FUNCTION_BLOCK PIDMgr3 (* Basic Function Block Type *)
  (* Standard: 61499-2 *)
  (* Version 0.0, 9/5/2025, Schneider Electric, Template *)
  PACKAGE SE.Nereda;
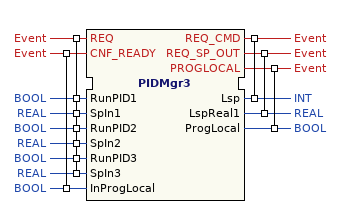
  EVENT_INPUT
    REQ WITH RunPID1, SpIn1, RunPID2, SpIn2, RunPID3, SpIn3; (* Normal Execution Request *)
    CNF_READY WITH InProgLocal;
  END_EVENT
  EVENT_OUTPUT
    REQ_CMD WITH Lsp;
    REQ_SP_OUT WITH LspReal1;
    PROGLOCAL WITH ProgLocal; (* Execution Confirmation *)
  END_EVENT
  VAR_INPUT
    RunPID1 : BOOL; (* Input event qualifier *)
    SpIn1 : REAL;
    RunPID2 : BOOL;
    SpIn2 : REAL;
    RunPID3 : BOOL;
    SpIn3 : REAL;
    InProgLocal : BOOL;
  END_VAR
  VAR_OUTPUT
    Lsp : INT;
    LspReal1 : REAL;
    ProgLocal : BOOL;
  END_VAR
  VAR
    InLsp : REAL;
  END_VAR
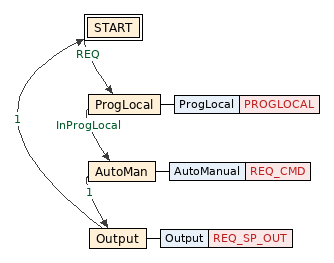
  EC_STATES
    START; (* Initial State *)
    ProgLocal : ProgLocal -> PROGLOCAL; (* Normal execution *)
    AutoMan : AutoManual -> REQ_CMD;
    Output : Output -> REQ_SP_OUT;
  END_STATES
  EC_TRANSITIONS
    START TO ProgLocal := REQ;
    ProgLocal TO AutoMan := InProgLocal;
    AutoMan TO Output := 1;
    Output TO START := 1;
  END_TRANSITIONS
  ALGORITHM ProgLocal IN ST: (* Normally executed algorithm *)
ProgLocal := TRUE;
  END_ALGORITHM
  ALGORITHM AutoManual IN ST: (* Put PID in AUTO or MANUAL *)
IF RunPID1 OR RunPID2 OR RunPID3 THEN
	Lsp := 1;
ELSE
	Lsp := 0;
END_IF;
  END_ALGORITHM
  ALGORITHM Output IN ST: (* Set output to 0 if off *)
InLsp := 0;

IF RunPID1 AND (SpIn1 > InLsp) THEN
    InLsp := SpIn1;
END_IF;

IF RunPID2 AND (SpIn2 > InLsp) THEN
    InLsp := SpIn2;
END_IF;

IF RunPID3 AND (SpIn3 > InLsp) THEN
    InLsp := SpIn3;
END_IF;

LspReal1 := InLsp;
  END_ALGORITHM
END_FUNCTION_BLOCK
